(* CoDeSys 2.3.9.37 project: Cap6_5.pro *)
(* Libraries: Standard.lib 4.10.05 12:14:46 *)

(* POU PLC_PRG, LD *)
PROGRAM PLC_PRG
VAR
	A: BOOL;
	Tiempo: TIME;
	B: BOOL;
	MiFlanco: R_TRIG;
	Contador: INT:=0;
	C: BOOL;
	Mitempo: TON;
	Salida: BOOL;
END_VAR
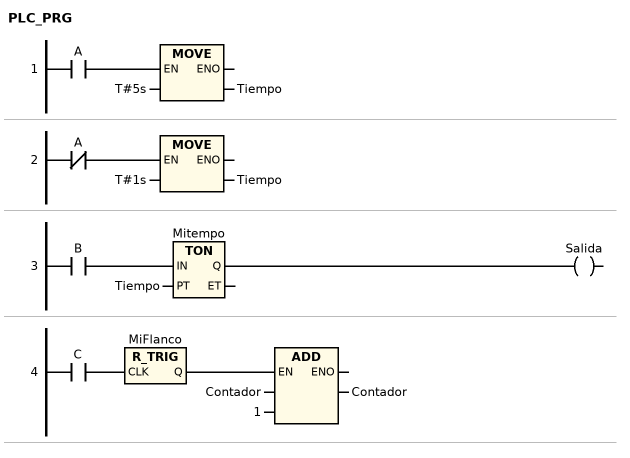
_LD_ (* Ladder Diagram *)
NETWORK 1
	[A]
		EN --- MOVE(T#5s) => Tiempo
NETWORK 2
	[/A]
		EN --- MOVE(T#1s) => Tiempo
NETWORK 3
	[B] - Mitempo:TON(IN: *, PT: Tiempo) --- (Salida)
NETWORK 4
	[C] - MiFlanco:R_TRIG(CLK: *)
		EN --- ADD(Contador, 1) => Contador
_END_LD_
(* the same logic as Structured Text *)
(* Network 1 *)
IF A THEN
	Tiempo := T#5s;
END_IF;
(* Network 2 *)
IF NOT A THEN
	Tiempo := T#1s;
END_IF;
(* Network 3 *)
Mitempo(IN := B, PT := Tiempo);
Salida := Mitempo.Q;
(* Network 4 *)
MiFlanco(CLK := C);
IF MiFlanco.Q THEN
	Contador := Contador + 1;
END_IF;
END_PROGRAM

(* Visualisation Visu
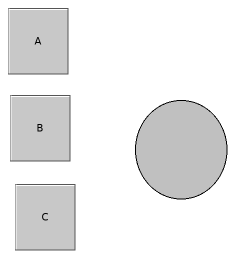
button at (43,29)-(103,95): text "A"; toggles PLC_PRG.A
button at (45,116)-(105,182): text "B"; toggles PLC_PRG.B
button at (50,205)-(110,271): text "C"; taps PLC_PRG.C
ellipse at (170,121)-(262,220): alarm colour if PLC_PRG.Salida
*)
